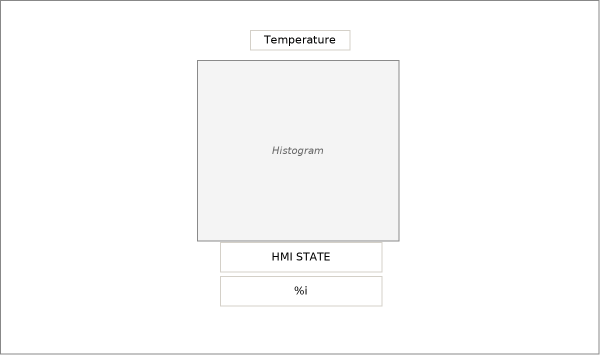
VISUALIZATION Set_Sensor  // 600x355
    Textfield (250,30 100x20), "Temperature"
    Textfield (220,242 162x30), "HMI STATE"
    Textfield (220,276 162x30), "%i", text variable: HMI_Global.HMI_State
    Histogram (197,60 202x181), scale format: %.1f, scale 0..100
        p1518820177: HMI_Global.HMI_IN_Temp
        p102497268: HMI_Global.HMI_IN_Temp
        p788070771: ARRAY [0..4] OF REAL
END_VISUALIZATION

(* stored: Version 1.1.0.1, ProductVersion 3.1.4024.12
   Visu Set_Sensor: Id {f3031d2d-57fd-49d1-9425-de7404289e92} *)
